// TIA Portal V16 export
// export: Created 2024-09-05T17:40:14.1588641Z, ExportSetting WithDefaults, DisplayName Totally Integrated Automation Portal, DisplayVersion V16 Update 6, DisplayName TIA Portal Version Control Interface, DisplayVersion V16 Update 2, DisplayName TIA Portal Openness, DisplayVersion V16 Update 6, DisplayName STEP 7 Professional, DisplayVersion V16 Update 6, DisplayName STEP 7 Safety, DisplayVersion V16, DisplayName WinCC Advanced, DisplayVersion V16 Update 6
TYPE "UDT_TurnTableOutputs"
// stored: IsFailsafeCompliant false
   STRUCT
      Enable : Bool;
      Stop : Bool;
      CycleCW : Bool;
      CycleCCW : Bool;
      JogCW : Bool;
      JogCCW : Bool;
      ResetError : Bool;
      WatchdogReceive : Bool;
   END_STRUCT;
END_TYPE
